FUNCTION_BLOCK Contactor
VAR
	output AT %Q*	:	BOOL;
END_VAR

METHOD PUBLIC SwitchOff
VAR_INPUT
END_VAR
output := FALSE;
END_METHOD

METHOD PUBLIC SwitchOn
VAR_INPUT
END_VAR
output := TRUE;
END_METHOD

END_FUNCTION_BLOCK

(* stored: Version 1.1.0.1, ProductVersion 3.1.4024.11
   POU Contactor: Id {9cdfaaab-0f05-497b-9988-34bbe645723a}, SpecialFunc None
   Method SwitchOff: Id {0f767173-681c-4ef9-b788-4b0fb4302ed0}
   Method SwitchOn: Id {f3b273df-0b8e-47b8-b7d0-3e6b4875561f} *)
